Staubli VAL3: saveInputOutput.pjx

--- saveInputOutput.pjx ---
Parameters version=s7.5 stackSize=5000 millimeterUnit=true
Program file=decompose_num.pgx
Program file=decompose_wait.pgx
Program file=getItem_num.pgx
Program file=getSize_num.pgx
Program file=getValue_num.pgx
Program file=get_num.pgx
Program file=insert_aCOunt.pgx
Program file=insert_aIn.pgx
Program file=insert_aOutput.pgx
Program file=insert_cCount.pgx
Program file=insert_dIn.pgx
Program file=insert_dOut.pgx
Program file=replaceIO.pgx
Program file=resetAll.pgx
Program file=setInput.pgx
Program file=setOutput.pgx
Data file=saveInputOutput.dtx
Type name=aioItem path=Disk://kernel/template/aioItem/aioItem.pjx
Type name=dioItem path=Disk://kernel/template/dioItem/dioItem.pjx
Type name=countItem path=Disk://kernel/template/countItem/countItem.pjx

--- saveInputOutput.dtx ---
public aio MbAnaIn[4]
  [0] = {link=ModbusSrv-0\Modbus-Word\MbAnaIn[0]}
  [1] = {link=ModbusSrv-0\Modbus-Word\MbAnaIn[1]}
  [2] = {link=ModbusSrv-0\Modbus-Word\MbAnaIn[2]}
  [3] = {link=ModbusSrv-0\Modbus-Word\MbAnaIn[3]}
public aio MbAnaOut[4]
  [0] = {link=ModbusSrv-0\Modbus-Word\MbAnaOut[0]}
  [1] = {link=ModbusSrv-0\Modbus-Word\MbAnaOut[1]}
  [2] = {link=ModbusSrv-0\Modbus-Word\MbAnaOut[2]}
  [3] = {link=ModbusSrv-0\Modbus-Word\MbAnaOut[3]}
aio aNull
public aio aUser[10]
public aio aio_in
public aio aio_out
public aio cAin0 = {link=Can-Aio\%IB7}
public aio cAin1 = {link=Can-Aio\%IB23}
public aio cAin2 = {link=Can-Aio\%IB39}
public aio cAin3 = {link=Can-Aio\%IB55}
aio cAout0
aio cAout1
aio cAout2
aio cAout3
public aioItem aCount{}
public aioItem aInput{}
public aioItem aOutput{}
public bool bArmIO
public bool bBio
public bool bCS8
public bool bMio
public countItem cCount{}
  [num0]
    bool bActive = true
    bool bEnable = true
    num nCount
    string sID = "num0"
    string sName = "num0"
  [num1]
    bool bActive = true
    bool bEnable = true
    num nCount
    string sID = "num1"
    string sName = "num1"
  [num2]
    bool bActive = true
    bool bEnable = true
    num nCount
    string sID = "num2"
    string sName = "num2"
  [num3]
    bool bActive = true
    bool bEnable = true
    num nCount
    string sID = "num3"
    string sName = "num3"
  [num4]
    bool bActive = true
    bool bEnable = true
    num nCount
    string sID = "num4"
    string sName = "num4"
  [num5]
    bool bActive = true
    bool bEnable = true
    num nCount
    string sID = "num5"
    string sName = "num5"
  [num6]
    bool bActive = true
    bool bEnable = true
    num nCount
    string sID = "num6"
    string sName = "num6"
  [num7]
    bool bActive = true
    bool bEnable = true
    num nCount
    string sID = "num7"
    string sName = "num7"
  [num8]
    bool bActive = true
    bool bEnable = true
    num nCount
    string sID = "num8"
    string sName = "num8"
  [num9]
    bool bActive = true
    bool bEnable = true
    num nCount
    string sID = "num9"
    string sName = "num9"
public dio MbIn[100]
  [0] = {link=ModbusSrv-0\Modbus-Bit\MbIn[0]}
  [1] = {link=ModbusSrv-0\Modbus-Bit\MbIn[1]}
  [2] = {link=ModbusSrv-0\Modbus-Bit\MbIn[2]}
  [3] = {link=ModbusSrv-0\Modbus-Bit\MbIn[3]}
  [4] = {link=ModbusSrv-0\Modbus-Bit\MbIn[4]}
  [5] = {link=ModbusSrv-0\Modbus-Bit\MbIn[5]}
  [6] = {link=ModbusSrv-0\Modbus-Bit\MbIn[6]}
  [7] = {link=ModbusSrv-0\Modbus-Bit\MbIn[7]}
  [8] = {link=ModbusSrv-0\Modbus-Bit\MbIn[8]}
  [9] = {link=ModbusSrv-0\Modbus-Bit\MbIn[9]}
  [10] = {link=ModbusSrv-0\Modbus-Bit\MbIn[10]}
  [11] = {link=ModbusSrv-0\Modbus-Bit\MbIn[11]}
  [12] = {link=ModbusSrv-0\Modbus-Bit\MbIn[12]}
  [13] = {link=ModbusSrv-0\Modbus-Bit\MbIn[13]}
  [14] = {link=ModbusSrv-0\Modbus-Bit\MbIn[14]}
  [15] = {link=ModbusSrv-0\Modbus-Bit\MbIn[15]}
  [16] = {link=ModbusSrv-0\Modbus-Bit\MbIn[16]}
  [17] = {link=ModbusSrv-0\Modbus-Bit\MbIn[17]}
  [18] = {link=ModbusSrv-0\Modbus-Bit\MbIn[18]}
  [19] = {link=ModbusSrv-0\Modbus-Bit\MbIn[19]}
  [20] = {link=ModbusSrv-0\Modbus-Bit\MbIn[20]}
  [21] = {link=ModbusSrv-0\Modbus-Bit\MbIn[21]}
  [22] = {link=ModbusSrv-0\Modbus-Bit\MbIn[22]}
  [23] = {link=ModbusSrv-0\Modbus-Bit\MbIn[23]}
  [24] = {link=ModbusSrv-0\Modbus-Bit\MbIn[24]}
  [25] = {link=ModbusSrv-0\Modbus-Bit\MbIn[25]}
  [26] = {link=ModbusSrv-0\Modbus-Bit\MbIn[26]}
  [27] = {link=ModbusSrv-0\Modbus-Bit\MbIn[27]}
  [28] = {link=ModbusSrv-0\Modbus-Bit\MbIn[28]}
  [29] = {link=ModbusSrv-0\Modbus-Bit\MbIn[29]}
  [30] = {link=ModbusSrv-0\Modbus-Bit\MbIn[30]}
  [31] = {link=ModbusSrv-0\Modbus-Bit\MbIn[31]}
  [32] = {link=ModbusSrv-0\Modbus-Bit\MbIn[32]}
  [33] = {link=ModbusSrv-0\Modbus-Bit\MbIn[33]}
  [34] = {link=ModbusSrv-0\Modbus-Bit\MbIn[34]}
  [35] = {link=ModbusSrv-0\Modbus-Bit\MbIn[35]}
  [36] = {link=ModbusSrv-0\Modbus-Bit\MbIn[36]}
  [37] = {link=ModbusSrv-0\Modbus-Bit\MbIn[37]}
  [38] = {link=ModbusSrv-0\Modbus-Bit\MbIn[38]}
  [39] = {link=ModbusSrv-0\Modbus-Bit\MbIn[39]}
  [40] = {link=ModbusSrv-0\Modbus-Bit\MbIn[40]}
  [41] = {link=ModbusSrv-0\Modbus-Bit\MbIn[41]}
  [42] = {link=ModbusSrv-0\Modbus-Bit\MbIn[42]}
  [43] = {link=ModbusSrv-0\Modbus-Bit\MbIn[43]}
  [44] = {link=ModbusSrv-0\Modbus-Bit\MbIn[44]}
  [45] = {link=ModbusSrv-0\Modbus-Bit\MbIn[45]}
  [46] = {link=ModbusSrv-0\Modbus-Bit\MbIn[46]}
  [47] = {link=ModbusSrv-0\Modbus-Bit\MbIn[47]}
  [48] = {link=ModbusSrv-0\Modbus-Bit\MbIn[48]}
  [49] = {link=ModbusSrv-0\Modbus-Bit\MbIn[49]}
  [50] = {link=ModbusSrv-0\Modbus-Bit\MbIn[50]}
  [51] = {link=ModbusSrv-0\Modbus-Bit\MbIn[51]}
  [52] = {link=ModbusSrv-0\Modbus-Bit\MbIn[52]}
  [53] = {link=ModbusSrv-0\Modbus-Bit\MbIn[53]}
  [54] = {link=ModbusSrv-0\Modbus-Bit\MbIn[54]}
  [55] = {link=ModbusSrv-0\Modbus-Bit\MbIn[55]}
  [56] = {link=ModbusSrv-0\Modbus-Bit\MbIn[56]}
  [57] = {link=ModbusSrv-0\Modbus-Bit\MbIn[57]}
  [58] = {link=ModbusSrv-0\Modbus-Bit\MbIn[58]}
  [59] = {link=ModbusSrv-0\Modbus-Bit\MbIn[59]}
  [60] = {link=ModbusSrv-0\Modbus-Bit\MbIn[60]}
  [61] = {link=ModbusSrv-0\Modbus-Bit\MbIn[61]}
  [62] = {link=ModbusSrv-0\Modbus-Bit\MbIn[62]}
  [63] = {link=ModbusSrv-0\Modbus-Bit\MbIn[63]}
  [64] = {link=ModbusSrv-0\Modbus-Bit\MbIn[64]}
  [65] = {link=ModbusSrv-0\Modbus-Bit\MbIn[65]}
  [66] = {link=ModbusSrv-0\Modbus-Bit\MbIn[66]}
  [67] = {link=ModbusSrv-0\Modbus-Bit\MbIn[67]}
  [68] = {link=ModbusSrv-0\Modbus-Bit\MbIn[68]}
  [69] = {link=ModbusSrv-0\Modbus-Bit\MbIn[69]}
  [70] = {link=ModbusSrv-0\Modbus-Bit\MbIn[70]}
  [71] = {link=ModbusSrv-0\Modbus-Bit\MbIn[71]}
  [72] = {link=ModbusSrv-0\Modbus-Bit\MbIn[72]}
  [73] = {link=ModbusSrv-0\Modbus-Bit\MbIn[73]}
  [74] = {link=ModbusSrv-0\Modbus-Bit\MbIn[74]}
  [75] = {link=ModbusSrv-0\Modbus-Bit\MbIn[75]}
  [76] = {link=ModbusSrv-0\Modbus-Bit\MbIn[76]}
  [77] = {link=ModbusSrv-0\Modbus-Bit\MbIn[77]}
  [78] = {link=ModbusSrv-0\Modbus-Bit\MbIn[78]}
  [79] = {link=ModbusSrv-0\Modbus-Bit\MbIn[79]}
  [80] = {link=ModbusSrv-0\Modbus-Bit\MbIn[80]}
  [81] = {link=ModbusSrv-0\Modbus-Bit\MbIn[81]}
  [82] = {link=ModbusSrv-0\Modbus-Bit\MbIn[82]}
  [83] = {link=ModbusSrv-0\Modbus-Bit\MbIn[83]}
  [84] = {link=ModbusSrv-0\Modbus-Bit\MbIn[84]}
  [85] = {link=ModbusSrv-0\Modbus-Bit\MbIn[85]}
  [86] = {link=ModbusSrv-0\Modbus-Bit\MbIn[86]}
  [87] = {link=ModbusSrv-0\Modbus-Bit\MbIn[87]}
  [88] = {link=ModbusSrv-0\Modbus-Bit\MbIn[88]}
  [89] = {link=ModbusSrv-0\Modbus-Bit\MbIn[89]}
  [90] = {link=ModbusSrv-0\Modbus-Bit\MbIn[90]}
  [91] = {link=ModbusSrv-0\Modbus-Bit\MbIn[91]}
  [92] = {link=ModbusSrv-0\Modbus-Bit\MbIn[92]}
  [93] = {link=ModbusSrv-0\Modbus-Bit\MbIn[93]}
  [94] = {link=ModbusSrv-0\Modbus-Bit\MbIn[94]}
  [95] = {link=ModbusSrv-0\Modbus-Bit\MbIn[95]}
  [96] = {link=ModbusSrv-0\Modbus-Bit\MbIn[96]}
  [97] = {link=ModbusSrv-0\Modbus-Bit\MbIn[97]}
  [98] = {link=ModbusSrv-0\Modbus-Bit\MbIn[98]}
  [99] = {link=ModbusSrv-0\Modbus-Bit\MbIn[99]}
public dio MbOut[100]
  [0] = {link=ModbusSrv-0\Modbus-Bit\MbOut[0]}
  [1] = {link=ModbusSrv-0\Modbus-Bit\MbOut[1]}
  [2] = {link=ModbusSrv-0\Modbus-Bit\MbOut[2]}
  [3] = {link=ModbusSrv-0\Modbus-Bit\MbOut[3]}
  [4] = {link=ModbusSrv-0\Modbus-Bit\MbOut[4]}
  [5] = {link=ModbusSrv-0\Modbus-Bit\MbOut[5]}
  [6] = {link=ModbusSrv-0\Modbus-Bit\MbOut[6]}
  [7] = {link=ModbusSrv-0\Modbus-Bit\MbOut[7]}
  [8] = {link=ModbusSrv-0\Modbus-Bit\MbOut[8]}
  [9] = {link=ModbusSrv-0\Modbus-Bit\MbOut[9]}
  [10] = {link=ModbusSrv-0\Modbus-Bit\MbOut[10]}
  [11] = {link=ModbusSrv-0\Modbus-Bit\MbOut[11]}
  [12] = {link=ModbusSrv-0\Modbus-Bit\MbOut[12]}
  [13] = {link=ModbusSrv-0\Modbus-Bit\MbOut[13]}
  [14] = {link=ModbusSrv-0\Modbus-Bit\MbOut[14]}
  [15] = {link=ModbusSrv-0\Modbus-Bit\MbOut[15]}
  [16] = {link=ModbusSrv-0\Modbus-Bit\MbOut[16]}
  [17] = {link=ModbusSrv-0\Modbus-Bit\MbOut[17]}
  [18] = {link=ModbusSrv-0\Modbus-Bit\MbOut[18]}
  [19] = {link=ModbusSrv-0\Modbus-Bit\MbOut[19]}
  [20] = {link=ModbusSrv-0\Modbus-Bit\MbOut[20]}
  [21] = {link=ModbusSrv-0\Modbus-Bit\MbOut[21]}
  [22] = {link=ModbusSrv-0\Modbus-Bit\MbOut[22]}
  [23] = {link=ModbusSrv-0\Modbus-Bit\MbOut[23]}
  [24] = {link=ModbusSrv-0\Modbus-Bit\MbOut[24]}
  [25] = {link=ModbusSrv-0\Modbus-Bit\MbOut[25]}
  [26] = {link=ModbusSrv-0\Modbus-Bit\MbOut[26]}
  [27] = {link=ModbusSrv-0\Modbus-Bit\MbOut[27]}
  [28] = {link=ModbusSrv-0\Modbus-Bit\MbOut[28]}
  [29] = {link=ModbusSrv-0\Modbus-Bit\MbOut[29]}
  [30] = {link=ModbusSrv-0\Modbus-Bit\MbOut[30]}
  [31] = {link=ModbusSrv-0\Modbus-Bit\MbOut[31]}
  [32] = {link=ModbusSrv-0\Modbus-Bit\MbOut[32]}
  [33] = {link=ModbusSrv-0\Modbus-Bit\MbOut[33]}
  [34] = {link=ModbusSrv-0\Modbus-Bit\MbOut[34]}
  [35] = {link=ModbusSrv-0\Modbus-Bit\MbOut[35]}
  [36] = {link=ModbusSrv-0\Modbus-Bit\MbOut[36]}
  [37] = {link=ModbusSrv-0\Modbus-Bit\MbOut[37]}
  [38] = {link=ModbusSrv-0\Modbus-Bit\MbOut[38]}
  [39] = {link=ModbusSrv-0\Modbus-Bit\MbOut[39]}
  [40] = {link=ModbusSrv-0\Modbus-Bit\MbOut[40]}
  [41] = {link=ModbusSrv-0\Modbus-Bit\MbOut[41]}
  [42] = {link=ModbusSrv-0\Modbus-Bit\MbOut[42]}
  [43] = {link=ModbusSrv-0\Modbus-Bit\MbOut[43]}
  [44] = {link=ModbusSrv-0\Modbus-Bit\MbOut[44]}
  [45] = {link=ModbusSrv-0\Modbus-Bit\MbOut[45]}
  [46] = {link=ModbusSrv-0\Modbus-Bit\MbOut[46]}
  [47] = {link=ModbusSrv-0\Modbus-Bit\MbOut[47]}
  [48] = {link=ModbusSrv-0\Modbus-Bit\MbOut[48]}
  [49] = {link=ModbusSrv-0\Modbus-Bit\MbOut[49]}
  [50] = {link=ModbusSrv-0\Modbus-Bit\MbOut[50]}
  [51] = {link=ModbusSrv-0\Modbus-Bit\MbOut[51]}
  [52] = {link=ModbusSrv-0\Modbus-Bit\MbOut[52]}
  [53] = {link=ModbusSrv-0\Modbus-Bit\MbOut[53]}
  [54] = {link=ModbusSrv-0\Modbus-Bit\MbOut[54]}
  [55] = {link=ModbusSrv-0\Modbus-Bit\MbOut[55]}
  [56] = {link=ModbusSrv-0\Modbus-Bit\MbOut[56]}
  [57] = {link=ModbusSrv-0\Modbus-Bit\MbOut[57]}
  [58] = {link=ModbusSrv-0\Modbus-Bit\MbOut[58]}
  [59] = {link=ModbusSrv-0\Modbus-Bit\MbOut[59]}
  [60] = {link=ModbusSrv-0\Modbus-Bit\MbOut[60]}
  [61] = {link=ModbusSrv-0\Modbus-Bit\MbOut[61]}
  [62] = {link=ModbusSrv-0\Modbus-Bit\MbOut[62]}
  [63] = {link=ModbusSrv-0\Modbus-Bit\MbOut[63]}
  [64] = {link=ModbusSrv-0\Modbus-Bit\MbOut[64]}
  [65] = {link=ModbusSrv-0\Modbus-Bit\MbOut[65]}
  [66] = {link=ModbusSrv-0\Modbus-Bit\MbOut[66]}
  [67] = {link=ModbusSrv-0\Modbus-Bit\MbOut[67]}
  [68] = {link=ModbusSrv-0\Modbus-Bit\MbOut[68]}
  [69] = {link=ModbusSrv-0\Modbus-Bit\MbOut[69]}
  [70] = {link=ModbusSrv-0\Modbus-Bit\MbOut[70]}
  [71] = {link=ModbusSrv-0\Modbus-Bit\MbOut[71]}
  [72] = {link=ModbusSrv-0\Modbus-Bit\MbOut[72]}
  [73] = {link=ModbusSrv-0\Modbus-Bit\MbOut[73]}
  [74] = {link=ModbusSrv-0\Modbus-Bit\MbOut[74]}
  [75] = {link=ModbusSrv-0\Modbus-Bit\MbOut[75]}
  [76] = {link=ModbusSrv-0\Modbus-Bit\MbOut[76]}
  [77] = {link=ModbusSrv-0\Modbus-Bit\MbOut[77]}
  [78] = {link=ModbusSrv-0\Modbus-Bit\MbOut[78]}
  [79] = {link=ModbusSrv-0\Modbus-Bit\MbOut[79]}
  [80] = {link=ModbusSrv-0\Modbus-Bit\MbOut[80]}
  [81] = {link=ModbusSrv-0\Modbus-Bit\MbOut[81]}
  [82] = {link=ModbusSrv-0\Modbus-Bit\MbOut[82]}
  [83] = {link=ModbusSrv-0\Modbus-Bit\MbOut[83]}
  [84] = {link=ModbusSrv-0\Modbus-Bit\MbOut[84]}
  [85] = {link=ModbusSrv-0\Modbus-Bit\MbOut[85]}
  [86] = {link=ModbusSrv-0\Modbus-Bit\MbOut[86]}
  [87] = {link=ModbusSrv-0\Modbus-Bit\MbOut[87]}
  [88] = {link=ModbusSrv-0\Modbus-Bit\MbOut[88]}
  [89] = {link=ModbusSrv-0\Modbus-Bit\MbOut[89]}
  [90] = {link=ModbusSrv-0\Modbus-Bit\MbOut[90]}
  [91] = {link=ModbusSrv-0\Modbus-Bit\MbOut[91]}
  [92] = {link=ModbusSrv-0\Modbus-Bit\MbOut[92]}
  [93] = {link=ModbusSrv-0\Modbus-Bit\MbOut[93]}
  [94] = {link=ModbusSrv-0\Modbus-Bit\MbOut[94]}
  [95] = {link=ModbusSrv-0\Modbus-Bit\MbOut[95]}
  [96] = {link=ModbusSrv-0\Modbus-Bit\MbOut[96]}
  [97] = {link=ModbusSrv-0\Modbus-Bit\MbOut[97]}
  [98] = {link=ModbusSrv-0\Modbus-Bit\MbOut[98]}
  [99] = {link=ModbusSrv-0\Modbus-Bit\MbOut[99]}
dio NetIn0 = {link=ApplicomIO-1\TOPIC1_A-BLOCKA\%I0}
dio NetIn1 = {link=ApplicomIO-1\TOPIC1_A-BLOCKA\%I1}
dio NetIn10 = {link=ApplicomIO-1\TOPIC1_A-BLOCKA\%I10}
dio NetIn11 = {link=ApplicomIO-1\TOPIC1_A-BLOCKA\%I11}
dio NetIn12 = {link=ApplicomIO-1\TOPIC1_A-BLOCKA\%I12}
dio NetIn13 = {link=ApplicomIO-1\TOPIC1_A-BLOCKA\%I13}
dio NetIn14 = {link=ApplicomIO-1\TOPIC1_A-BLOCKA\%I14}
dio NetIn15 = {link=ApplicomIO-1\TOPIC1_A-BLOCKA\%I15}
dio NetIn16 = {link=ApplicomIO-1\TOPIC1_A-BLOCKA\%I16}
dio NetIn17 = {link=ApplicomIO-1\TOPIC1_A-BLOCKA\%I17}
dio NetIn18 = {link=ApplicomIO-1\TOPIC1_A-BLOCKA\%I18}
dio NetIn19 = {link=ApplicomIO-1\TOPIC1_A-BLOCKA\%I19}
dio NetIn2 = {link=ApplicomIO-1\TOPIC1_A-BLOCKA\%I2}
dio NetIn20 = {link=ApplicomIO-1\TOPIC1_A-BLOCKA\%I20}
dio NetIn21 = {link=ApplicomIO-1\TOPIC1_A-BLOCKA\%I21}
dio NetIn22 = {link=ApplicomIO-1\TOPIC1_A-BLOCKA\%I22}
dio NetIn23 = {link=ApplicomIO-1\TOPIC1_A-BLOCKA\%I23}
dio NetIn24 = {link=ApplicomIO-1\TOPIC1_A-BLOCKA\%I24}
dio NetIn25 = {link=ApplicomIO-1\TOPIC1_A-BLOCKA\%I25}
dio NetIn26 = {link=ApplicomIO-1\TOPIC1_A-BLOCKA\%I26}
dio NetIn27 = {link=ApplicomIO-1\TOPIC1_A-BLOCKA\%I27}
dio NetIn28 = {link=ApplicomIO-1\TOPIC1_A-BLOCKA\%I28}
dio NetIn29 = {link=ApplicomIO-1\TOPIC1_A-BLOCKA\%I29}
dio NetIn3 = {link=ApplicomIO-1\TOPIC1_A-BLOCKA\%I3}
dio NetIn30 = {link=ApplicomIO-1\TOPIC1_A-BLOCKA\%I30}
dio NetIn31 = {link=ApplicomIO-1\TOPIC1_A-BLOCKA\%I31}
dio NetIn32 = {link=ApplicomIO-1\TOPIC1_A-BLOCKA\%I32}
dio NetIn33 = {link=ApplicomIO-1\TOPIC1_A-BLOCKA\%I33}
dio NetIn34 = {link=ApplicomIO-1\TOPIC1_A-BLOCKA\%I34}
dio NetIn35 = {link=ApplicomIO-1\TOPIC1_A-BLOCKA\%I35}
dio NetIn36 = {link=ApplicomIO-1\TOPIC1_A-BLOCKA\%I36}
dio NetIn37 = {link=ApplicomIO-1\TOPIC1_A-BLOCKA\%I37}
dio NetIn38 = {link=ApplicomIO-1\TOPIC1_A-BLOCKA\%I38}
dio NetIn39 = {link=ApplicomIO-1\TOPIC1_A-BLOCKA\%I39}
dio NetIn4 = {link=ApplicomIO-1\TOPIC1_A-BLOCKA\%I4}
dio NetIn40 = {link=ApplicomIO-1\TOPIC1_A-BLOCKA\%I40}
dio NetIn41 = {link=ApplicomIO-1\TOPIC1_A-BLOCKA\%I41}
dio NetIn42 = {link=ApplicomIO-1\TOPIC1_A-BLOCKA\%I42}
dio NetIn43 = {link=ApplicomIO-1\TOPIC1_A-BLOCKA\%I43}
dio NetIn44 = {link=ApplicomIO-1\TOPIC1_A-BLOCKA\%I44}
dio NetIn45 = {link=ApplicomIO-1\TOPIC1_A-BLOCKA\%I45}
dio NetIn46 = {link=ApplicomIO-1\TOPIC1_A-BLOCKA\%I46}
dio NetIn47 = {link=ApplicomIO-1\TOPIC1_A-BLOCKA\%I47}
dio NetIn48 = {link=ApplicomIO-1\TOPIC1_A-BLOCKA\%I48}
dio NetIn49 = {link=ApplicomIO-1\TOPIC1_A-BLOCKA\%I49}
dio NetIn5 = {link=ApplicomIO-1\TOPIC1_A-BLOCKA\%I5}
dio NetIn50 = {link=ApplicomIO-1\TOPIC1_A-BLOCKA\%I50}
dio NetIn51 = {link=ApplicomIO-1\TOPIC1_A-BLOCKA\%I51}
dio NetIn52 = {link=ApplicomIO-1\TOPIC1_A-BLOCKA\%I52}
dio NetIn53 = {link=ApplicomIO-1\TOPIC1_A-BLOCKA\%I53}
dio NetIn54 = {link=ApplicomIO-1\TOPIC1_A-BLOCKA\%I54}
dio NetIn55 = {link=ApplicomIO-1\TOPIC1_A-BLOCKA\%I55}
dio NetIn56 = {link=ApplicomIO-1\TOPIC1_A-BLOCKA\%I56}
dio NetIn57 = {link=ApplicomIO-1\TOPIC1_A-BLOCKA\%I57}
dio NetIn58 = {link=ApplicomIO-1\TOPIC1_A-BLOCKA\%I58}
dio NetIn59 = {link=ApplicomIO-1\TOPIC1_A-BLOCKA\%I59}
dio NetIn6 = {link=ApplicomIO-1\TOPIC1_A-BLOCKA\%I6}
dio NetIn60 = {link=ApplicomIO-1\TOPIC1_A-BLOCKA\%I60}
dio NetIn61 = {link=ApplicomIO-1\TOPIC1_A-BLOCKA\%I61}
dio NetIn62 = {link=ApplicomIO-1\TOPIC1_A-BLOCKA\%I62}
dio NetIn63 = {link=ApplicomIO-1\TOPIC1_A-BLOCKA\%I63}
dio NetIn7 = {link=ApplicomIO-1\TOPIC1_A-BLOCKA\%I7}
dio NetIn8 = {link=ApplicomIO-1\TOPIC1_A-BLOCKA\%I8}
dio NetIn9 = {link=ApplicomIO-1\TOPIC1_A-BLOCKA\%I9}
dio NetOut0 = {link=ApplicomIO-1\TOPIC1_A-BLOCKA\%Q0}
dio NetOut1 = {link=ApplicomIO-1\TOPIC1_A-BLOCKA\%Q1}
dio NetOut10 = {link=ApplicomIO-1\TOPIC1_A-BLOCKA\%Q10}
dio NetOut11 = {link=ApplicomIO-1\TOPIC1_A-BLOCKA\%Q11}
dio NetOut12 = {link=ApplicomIO-1\TOPIC1_A-BLOCKA\%Q12}
dio NetOut13 = {link=ApplicomIO-1\TOPIC1_A-BLOCKA\%Q13}
dio NetOut14 = {link=ApplicomIO-1\TOPIC1_A-BLOCKA\%Q14}
dio NetOut15 = {link=ApplicomIO-1\TOPIC1_A-BLOCKA\%Q15}
dio NetOut16 = {link=ApplicomIO-1\TOPIC1_A-BLOCKA\%Q16}
dio NetOut17 = {link=ApplicomIO-1\TOPIC1_A-BLOCKA\%Q17}
dio NetOut18 = {link=ApplicomIO-1\TOPIC1_A-BLOCKA\%Q18}
dio NetOut19 = {link=ApplicomIO-1\TOPIC1_A-BLOCKA\%Q19}
dio NetOut2 = {link=ApplicomIO-1\TOPIC1_A-BLOCKA\%Q2}
dio NetOut20 = {link=ApplicomIO-1\TOPIC1_A-BLOCKA\%Q20}
dio NetOut21 = {link=ApplicomIO-1\TOPIC1_A-BLOCKA\%Q21}
dio NetOut22 = {link=ApplicomIO-1\TOPIC1_A-BLOCKA\%Q22}
dio NetOut23 = {link=ApplicomIO-1\TOPIC1_A-BLOCKA\%Q23}
dio NetOut24 = {link=ApplicomIO-1\TOPIC1_A-BLOCKA\%Q24}
dio NetOut25 = {link=ApplicomIO-1\TOPIC1_A-BLOCKA\%Q25}
dio NetOut26 = {link=ApplicomIO-1\TOPIC1_A-BLOCKA\%Q26}
dio NetOut27 = {link=ApplicomIO-1\TOPIC1_A-BLOCKA\%Q27}
dio NetOut28 = {link=ApplicomIO-1\TOPIC1_A-BLOCKA\%Q28}
dio NetOut29 = {link=ApplicomIO-1\TOPIC1_A-BLOCKA\%Q29}
dio NetOut3 = {link=ApplicomIO-1\TOPIC1_A-BLOCKA\%Q3}
dio NetOut30 = {link=ApplicomIO-1\TOPIC1_A-BLOCKA\%Q30}
dio NetOut31 = {link=ApplicomIO-1\TOPIC1_A-BLOCKA\%Q31}
dio NetOut32 = {link=ApplicomIO-1\TOPIC1_A-BLOCKA\%Q32}
dio NetOut33 = {link=ApplicomIO-1\TOPIC1_A-BLOCKA\%Q33}
dio NetOut34 = {link=ApplicomIO-1\TOPIC1_A-BLOCKA\%Q34}
dio NetOut35 = {link=ApplicomIO-1\TOPIC1_A-BLOCKA\%Q35}
dio NetOut36 = {link=ApplicomIO-1\TOPIC1_A-BLOCKA\%Q36}
dio NetOut37 = {link=ApplicomIO-1\TOPIC1_A-BLOCKA\%Q37}
dio NetOut38 = {link=ApplicomIO-1\TOPIC1_A-BLOCKA\%Q38}
dio NetOut39 = {link=ApplicomIO-1\TOPIC1_A-BLOCKA\%Q39}
dio NetOut4 = {link=ApplicomIO-1\TOPIC1_A-BLOCKA\%Q4}
dio NetOut40 = {link=ApplicomIO-1\TOPIC1_A-BLOCKA\%Q40}
dio NetOut41 = {link=ApplicomIO-1\TOPIC1_A-BLOCKA\%Q41}
dio NetOut42 = {link=ApplicomIO-1\TOPIC1_A-BLOCKA\%Q42}
dio NetOut43 = {link=ApplicomIO-1\TOPIC1_A-BLOCKA\%Q43}
dio NetOut44 = {link=ApplicomIO-1\TOPIC1_A-BLOCKA\%Q44}
dio NetOut45 = {link=ApplicomIO-1\TOPIC1_A-BLOCKA\%Q45}
dio NetOut46 = {link=ApplicomIO-1\TOPIC1_A-BLOCKA\%Q46}
dio NetOut47 = {link=ApplicomIO-1\TOPIC1_A-BLOCKA\%Q47}
dio NetOut48 = {link=ApplicomIO-1\TOPIC1_A-BLOCKA\%Q48}
dio NetOut49 = {link=ApplicomIO-1\TOPIC1_A-BLOCKA\%Q49}
dio NetOut5 = {link=ApplicomIO-1\TOPIC1_A-BLOCKA\%Q5}
dio NetOut50 = {link=ApplicomIO-1\TOPIC1_A-BLOCKA\%Q50}
dio NetOut51 = {link=ApplicomIO-1\TOPIC1_A-BLOCKA\%Q51}
dio NetOut52 = {link=ApplicomIO-1\TOPIC1_A-BLOCKA\%Q52}
dio NetOut53 = {link=ApplicomIO-1\TOPIC1_A-BLOCKA\%Q53}
dio NetOut54 = {link=ApplicomIO-1\TOPIC1_A-BLOCKA\%Q54}
dio NetOut55 = {link=ApplicomIO-1\TOPIC1_A-BLOCKA\%Q55}
dio NetOut56 = {link=ApplicomIO-1\TOPIC1_A-BLOCKA\%Q56}
dio NetOut57 = {link=ApplicomIO-1\TOPIC1_A-BLOCKA\%Q57}
dio NetOut58 = {link=ApplicomIO-1\TOPIC1_A-BLOCKA\%Q58}
dio NetOut59 = {link=ApplicomIO-1\TOPIC1_A-BLOCKA\%Q59}
dio NetOut6 = {link=ApplicomIO-1\TOPIC1_A-BLOCKA\%Q6}
dio NetOut60 = {link=ApplicomIO-1\TOPIC1_A-BLOCKA\%Q60}
dio NetOut61 = {link=ApplicomIO-1\TOPIC1_A-BLOCKA\%Q61}
dio NetOut62 = {link=ApplicomIO-1\TOPIC1_A-BLOCKA\%Q62}
dio NetOut63 = {link=ApplicomIO-1\TOPIC1_A-BLOCKA\%Q63}
dio NetOut7 = {link=ApplicomIO-1\TOPIC1_A-BLOCKA\%Q7}
dio NetOut8 = {link=ApplicomIO-1\TOPIC1_A-BLOCKA\%Q8}
dio NetOut9 = {link=ApplicomIO-1\TOPIC1_A-BLOCKA\%Q9}
public dio b2In0 = {link=BasicIO-2\%I0}
public dio b2In1 = {link=BasicIO-2\%I1}
public dio b2In10 = {link=BasicIO-2\%I10}
public dio b2In11 = {link=BasicIO-2\%I11}
public dio b2In12 = {link=BasicIO-2\%I12}
public dio b2In13 = {link=BasicIO-2\%I13}
public dio b2In14 = {link=BasicIO-2\%I14}
public dio b2In15 = {link=BasicIO-2\%I15}
public dio b2In2 = {link=BasicIO-2\%I2}
public dio b2In3 = {link=BasicIO-2\%I3}
public dio b2In4 = {link=BasicIO-2\%I4}
public dio b2In5 = {link=BasicIO-2\%I5}
public dio b2In6 = {link=BasicIO-2\%I6}
public dio b2In7 = {link=BasicIO-2\%I7}
public dio b2In8 = {link=BasicIO-2\%I8}
public dio b2In9 = {link=BasicIO-2\%I9}
public dio b2Out0 = {link=BasicIO-2\%Q0}
public dio b2Out1 = {link=BasicIO-2\%Q1}
public dio b2Out10 = {link=BasicIO-2\%Q10}
public dio b2Out11 = {link=BasicIO-2\%Q11}
public dio b2Out12 = {link=BasicIO-2\%Q12}
public dio b2Out13 = {link=BasicIO-2\%Q13}
public dio b2Out14 = {link=BasicIO-2\%Q14}
public dio b2Out15 = {link=BasicIO-2\%Q15}
public dio b2Out2 = {link=BasicIO-2\%Q2}
public dio b2Out3 = {link=BasicIO-2\%Q3}
public dio b2Out4 = {link=BasicIO-2\%Q4}
public dio b2Out5 = {link=BasicIO-2\%Q5}
public dio b2Out6 = {link=BasicIO-2\%Q6}
public dio b2Out7 = {link=BasicIO-2\%Q7}
public dio b2Out8 = {link=BasicIO-2\%Q8}
public dio b2Out9 = {link=BasicIO-2\%Q9}
public dio bIn0 = {link=BasicIO-1\%I0}
public dio bIn1 = {link=BasicIO-1\%I1}
public dio bIn10 = {link=BasicIO-1\%I10}
public dio bIn11 = {link=BasicIO-1\%I11}
public dio bIn12 = {link=BasicIO-1\%I12}
public dio bIn13 = {link=BasicIO-1\%I13}
public dio bIn14 = {link=BasicIO-1\%I14}
public dio bIn15 = {link=BasicIO-1\%I15}
public dio bIn2 = {link=BasicIO-1\%I2}
public dio bIn3 = {link=BasicIO-1\%I3}
public dio bIn4 = {link=BasicIO-1\%I4}
public dio bIn5 = {link=BasicIO-1\%I5}
public dio bIn6 = {link=BasicIO-1\%I6}
public dio bIn7 = {link=BasicIO-1\%I7}
public dio bIn8 = {link=BasicIO-1\%I8}
public dio bIn9 = {link=BasicIO-1\%I9}
public dio bOut0 = {link=BasicIO-1\%Q0}
public dio bOut1 = {link=BasicIO-1\%Q1}
public dio bOut10 = {link=BasicIO-1\%Q10}
public dio bOut11 = {link=BasicIO-1\%Q11}
public dio bOut12 = {link=BasicIO-1\%Q12}
public dio bOut13 = {link=BasicIO-1\%Q13}
public dio bOut14 = {link=BasicIO-1\%Q14}
public dio bOut15 = {link=BasicIO-1\%Q15}
public dio bOut2 = {link=BasicIO-1\%Q2}
public dio bOut3 = {link=BasicIO-1\%Q3}
public dio bOut4 = {link=BasicIO-1\%Q4}
public dio bOut5 = {link=BasicIO-1\%Q5}
public dio bOut6 = {link=BasicIO-1\%Q6}
public dio bOut7 = {link=BasicIO-1\%Q7}
public dio bOut8 = {link=BasicIO-1\%Q8}
public dio bOut9 = {link=BasicIO-1\%Q9}
public dio cDin0 = {link=Can-Dio\%I0}
public dio cDin1 = {link=Can-Dio\%I1}
public dio cDin2 = {link=Can-Dio\%I2}
public dio cDin3 = {link=Can-Dio\%I3}
public dio cDin4 = {link=Can-Dio\%I4}
public dio cDin5 = {link=Can-Dio\%I5}
public dio cDin6 = {link=Can-Dio\%I6}
public dio cDin7 = {link=Can-Dio\%I7}
public dio cDout0 = {link=Can-Dio\%Q0}
public dio cDout1 = {link=Can-Dio\%Q1}
public dio cDout2 = {link=Can-Dio\%Q2}
public dio cDout3 = {link=Can-Dio\%Q3}
public dio cDout4 = {link=Can-Dio\%Q4}
public dio cDout5 = {link=Can-Dio\%Q5}
public dio cDout6 = {link=Can-Dio\%Q6}
public dio cDout7 = {link=Can-Dio\%Q7}
public dio dInUser
dio dNull
public dio dOutUser
public dio fIn0 = {link=fIn0}
public dio fIn1 = {link=fIn1}
public dio fOut0 = {link=fOut0}
public dio mIn0 = {link=ModuleIO\%I0}
public dio mIn1 = {link=ModuleIO\%I1}
public dio mIn10 = {link=ModuleIO\%I10}
public dio mIn11 = {link=ModuleIO\%I11}
public dio mIn12 = {link=ModuleIO\%I12}
public dio mIn13 = {link=ModuleIO\%I13}
public dio mIn14 = {link=ModuleIO\%I14}
public dio mIn15 = {link=ModuleIO\%I15}
public dio mIn16 = {link=ModuleIO\%I16}
public dio mIn17 = {link=ModuleIO\%I17}
public dio mIn18 = {link=ModuleIO\%I18}
public dio mIn19 = {link=ModuleIO\%I19}
public dio mIn2 = {link=ModuleIO\%I2}
public dio mIn20 = {link=ModuleIO\%I20}
public dio mIn21 = {link=ModuleIO\%I21}
public dio mIn22 = {link=ModuleIO\%I22}
public dio mIn23 = {link=ModuleIO\%I23}
public dio mIn24 = {link=ModuleIO\%I24}
public dio mIn25 = {link=ModuleIO\%I25}
public dio mIn26 = {link=ModuleIO\%I26}
public dio mIn27 = {link=ModuleIO\%I27}
public dio mIn28 = {link=ModuleIO\%I28}
public dio mIn29 = {link=ModuleIO\%I29}
public dio mIn3 = {link=ModuleIO\%I3}
public dio mIn30 = {link=ModuleIO\%I30}
public dio mIn31 = {link=ModuleIO\%I31}
public dio mIn4 = {link=ModuleIO\%I4}
public dio mIn5 = {link=ModuleIO\%I5}
public dio mIn6 = {link=ModuleIO\%I6}
public dio mIn7 = {link=ModuleIO\%I7}
public dio mIn8 = {link=ModuleIO\%I8}
public dio mIn9 = {link=ModuleIO\%I9}
public dio mOut0 = {link=ModuleIO\%Q0}
public dio mOut1 = {link=ModuleIO\%Q1}
public dio mOut10 = {link=ModuleIO\%Q10}
public dio mOut11 = {link=ModuleIO\%Q11}
public dio mOut12 = {link=ModuleIO\%Q12}
public dio mOut13 = {link=ModuleIO\%Q13}
public dio mOut14 = {link=ModuleIO\%Q14}
public dio mOut15 = {link=ModuleIO\%Q15}
public dio mOut16 = {link=ModuleIO\%Q16}
public dio mOut17 = {link=ModuleIO\%Q17}
public dio mOut18 = {link=ModuleIO\%Q18}
public dio mOut19 = {link=ModuleIO\%Q19}
public dio mOut2 = {link=ModuleIO\%Q2}
public dio mOut20 = {link=ModuleIO\%Q20}
public dio mOut21 = {link=ModuleIO\%Q21}
public dio mOut22 = {link=ModuleIO\%Q22}
public dio mOut23 = {link=ModuleIO\%Q23}
public dio mOut24 = {link=ModuleIO\%Q24}
public dio mOut25 = {link=ModuleIO\%Q25}
public dio mOut26 = {link=ModuleIO\%Q26}
public dio mOut27 = {link=ModuleIO\%Q27}
public dio mOut28 = {link=ModuleIO\%Q28}
public dio mOut29 = {link=ModuleIO\%Q29}
public dio mOut3 = {link=ModuleIO\%Q3}
public dio mOut30 = {link=ModuleIO\%Q30}
public dio mOut31 = {link=ModuleIO\%Q31}
public dio mOut4 = {link=ModuleIO\%Q4}
public dio mOut5 = {link=ModuleIO\%Q5}
public dio mOut6 = {link=ModuleIO\%Q6}
public dio mOut7 = {link=ModuleIO\%Q7}
public dio mOut8 = {link=ModuleIO\%Q8}
public dio mOut9 = {link=ModuleIO\%Q9}
public dio usrIn0 = {link=usrIn0}
public dio usrIn1 = {link=usrIn1}
public dio valve1 = {link=valve1}
public dio valve2 = {link=valve2}
public dioItem dInput{}
  [NetIn00]
    bool bActive
    bool bEnable = true
    dio dDio = {link=ApplicomIO-1\TOPIC1_A-BLOCKA\%I0}
    string sID = "NetIn00"
    string sName = "NetIn00"
  [NetIn01]
    bool bActive
    bool bEnable = true
    dio dDio = {link=ApplicomIO-1\TOPIC1_A-BLOCKA\%I1}
    string sID = "NetIn01"
    string sName = "NetIn01"
  [NetIn02]
    bool bActive
    bool bEnable = true
    dio dDio = {link=ApplicomIO-1\TOPIC1_A-BLOCKA\%I2}
    string sID = "NetIn02"
    string sName = "NetIn02"
  [NetIn03]
    bool bActive
    bool bEnable = true
    dio dDio = {link=ApplicomIO-1\TOPIC1_A-BLOCKA\%I3}
    string sID = "NetIn03"
    string sName = "NetIn03"
  [NetIn04]
    bool bActive
    bool bEnable = true
    dio dDio = {link=ApplicomIO-1\TOPIC1_A-BLOCKA\%I4}
    string sID = "NetIn04"
    string sName = "NetIn04"
  [NetIn05]
    bool bActive
    bool bEnable = true
    dio dDio = {link=ApplicomIO-1\TOPIC1_A-BLOCKA\%I5}
    string sID = "NetIn05"
    string sName = "NetIn05"
  [NetIn06]
    bool bActive
    bool bEnable = true
    dio dDio = {link=ApplicomIO-1\TOPIC1_A-BLOCKA\%I6}
    string sID = "NetIn06"
    string sName = "NetIn06"
  [NetIn07]
    bool bActive
    bool bEnable = true
    dio dDio = {link=ApplicomIO-1\TOPIC1_A-BLOCKA\%I7}
    string sID = "NetIn07"
    string sName = "NetIn07"
  [NetIn08]
    bool bActive
    bool bEnable = true
    dio dDio = {link=ApplicomIO-1\TOPIC1_A-BLOCKA\%I8}
    string sID = "NetIn08"
    string sName = "NetIn08"
  [NetIn09]
    bool bActive
    bool bEnable = true
    dio dDio = {link=ApplicomIO-1\TOPIC1_A-BLOCKA\%I9}
    string sID = "NetIn09"
    string sName = "NetIn09"
  [NetIn10]
    bool bActive
    bool bEnable = true
    dio dDio = {link=ApplicomIO-1\TOPIC1_A-BLOCKA\%I10}
    string sID = "NetIn10"
    string sName = "NetIn10"
  [NetIn11]
    bool bActive
    bool bEnable = true
    dio dDio = {link=ApplicomIO-1\TOPIC1_A-BLOCKA\%I11}
    string sID = "NetIn11"
    string sName = "NetIn11"
  [NetIn12]
    bool bActive
    bool bEnable = true
    dio dDio = {link=ApplicomIO-1\TOPIC1_A-BLOCKA\%I12}
    string sID = "NetIn12"
    string sName = "NetIn12"
  [NetIn13]
    bool bActive
    bool bEnable = true
    dio dDio = {link=ApplicomIO-1\TOPIC1_A-BLOCKA\%I13}
    string sID = "NetIn13"
    string sName = "NetIn13"
  [NetIn14]
    bool bActive
    bool bEnable = true
    dio dDio = {link=ApplicomIO-1\TOPIC1_A-BLOCKA\%I14}
    string sID = "NetIn14"
    string sName = "NetIn14"
  [NetIn15]
    bool bActive
    bool bEnable = true
    dio dDio = {link=ApplicomIO-1\TOPIC1_A-BLOCKA\%I15}
    string sID = "NetIn15"
    string sName = "NetIn15"
  [NetIn16]
    bool bActive
    bool bEnable = true
    dio dDio = {link=ApplicomIO-1\TOPIC1_A-BLOCKA\%I16}
    string sID = "NetIn16"
    string sName = "NetIn16"
  [NetIn17]
    bool bActive
    bool bEnable = true
    dio dDio = {link=ApplicomIO-1\TOPIC1_A-BLOCKA\%I17}
    string sID = "NetIn17"
    string sName = "NetIn17"
  [NetIn18]
    bool bActive
    bool bEnable = true
    dio dDio = {link=ApplicomIO-1\TOPIC1_A-BLOCKA\%I18}
    string sID = "NetIn18"
    string sName = "NetIn18"
  [NetIn19]
    bool bActive
    bool bEnable = true
    dio dDio = {link=ApplicomIO-1\TOPIC1_A-BLOCKA\%I19}
    string sID = "NetIn19"
    string sName = "NetIn19"
  [NetIn20]
    bool bActive
    bool bEnable = true
    dio dDio = {link=ApplicomIO-1\TOPIC1_A-BLOCKA\%I20}
    string sID = "NetIn20"
    string sName = "NetIn20"
  [NetIn21]
    bool bActive
    bool bEnable = true
    dio dDio = {link=ApplicomIO-1\TOPIC1_A-BLOCKA\%I21}
    string sID = "NetIn21"
    string sName = "NetIn21"
  [NetIn22]
    bool bActive
    bool bEnable = true
    dio dDio = {link=ApplicomIO-1\TOPIC1_A-BLOCKA\%I22}
    string sID = "NetIn22"
    string sName = "NetIn22"
  [NetIn23]
    bool bActive
    bool bEnable = true
    dio dDio = {link=ApplicomIO-1\TOPIC1_A-BLOCKA\%I23}
    string sID = "NetIn23"
    string sName = "NetIn23"
  [NetIn24]
    bool bActive
    bool bEnable = true
    dio dDio = {link=ApplicomIO-1\TOPIC1_A-BLOCKA\%I24}
    string sID = "NetIn24"
    string sName = "NetIn24"
  [NetIn25]
    bool bActive
    bool bEnable = true
    dio dDio = {link=ApplicomIO-1\TOPIC1_A-BLOCKA\%I25}
    string sID = "NetIn25"
    string sName = "NetIn25"
  [NetIn26]
    bool bActive
    bool bEnable = true
    dio dDio = {link=ApplicomIO-1\TOPIC1_A-BLOCKA\%I26}
    string sID = "NetIn26"
    string sName = "NetIn26"
  [NetIn27]
    bool bActive
    bool bEnable = true
    dio dDio = {link=ApplicomIO-1\TOPIC1_A-BLOCKA\%I27}
    string sID = "NetIn27"
    string sName = "NetIn27"
  [NetIn28]
    bool bActive
    bool bEnable = true
    dio dDio = {link=ApplicomIO-1\TOPIC1_A-BLOCKA\%I28}
    string sID = "NetIn28"
    string sName = "NetIn28"
  [NetIn29]
    bool bActive
    bool bEnable = true
    dio dDio = {link=ApplicomIO-1\TOPIC1_A-BLOCKA\%I29}
    string sID = "NetIn29"
    string sName = "NetIn29"
  [NetIn30]
    bool bActive
    bool bEnable = true
    dio dDio = {link=ApplicomIO-1\TOPIC1_A-BLOCKA\%I30}
    string sID = "NetIn30"
    string sName = "NetIn30"
  [NetIn31]
    bool bActive
    bool bEnable = true
    dio dDio = {link=ApplicomIO-1\TOPIC1_A-BLOCKA\%I31}
    string sID = "NetIn31"
    string sName = "NetIn31"
  [NetIn32]
    bool bActive
    bool bEnable = true
    dio dDio = {link=ApplicomIO-1\TOPIC1_A-BLOCKA\%I32}
    string sID = "NetIn32"
    string sName = "NetIn32"
  [NetIn33]
    bool bActive
    bool bEnable = true
    dio dDio = {link=ApplicomIO-1\TOPIC1_A-BLOCKA\%I33}
    string sID = "NetIn33"
    string sName = "NetIn33"
  [NetIn34]
    bool bActive
    bool bEnable = true
    dio dDio = {link=ApplicomIO-1\TOPIC1_A-BLOCKA\%I34}
    string sID = "NetIn34"
    string sName = "NetIn34"
  [NetIn35]
    bool bActive
    bool bEnable = true
    dio dDio = {link=ApplicomIO-1\TOPIC1_A-BLOCKA\%I35}
    string sID = "NetIn35"
    string sName = "NetIn35"
  [NetIn36]
    bool bActive
    bool bEnable = true
    dio dDio = {link=ApplicomIO-1\TOPIC1_A-BLOCKA\%I36}
    string sID = "NetIn36"
    string sName = "NetIn36"
  [NetIn37]
    bool bActive
    bool bEnable = true
    dio dDio = {link=ApplicomIO-1\TOPIC1_A-BLOCKA\%I37}
    string sID = "NetIn37"
    string sName = "NetIn37"
  [NetIn38]
    bool bActive
    bool bEnable = true
    dio dDio = {link=ApplicomIO-1\TOPIC1_A-BLOCKA\%I38}
    string sID = "NetIn38"
    string sName = "NetIn38"
  [NetIn39]
    bool bActive
    bool bEnable = true
    dio dDio = {link=ApplicomIO-1\TOPIC1_A-BLOCKA\%I39}
    string sID = "NetIn39"
    string sName = "NetIn39"
  [NetIn40]
    bool bActive
    bool bEnable = true
    dio dDio = {link=ApplicomIO-1\TOPIC1_A-BLOCKA\%I40}
    string sID = "NetIn40"
    string sName = "NetIn40"
  [NetIn41]
    bool bActive
    bool bEnable = true
    dio dDio = {link=ApplicomIO-1\TOPIC1_A-BLOCKA\%I41}
    string sID = "NetIn41"
    string sName = "NetIn41"
  [NetIn42]
    bool bActive
    bool bEnable = true
    dio dDio = {link=ApplicomIO-1\TOPIC1_A-BLOCKA\%I42}
    string sID = "NetIn42"
    string sName = "NetIn42"
  [NetIn43]
    bool bActive
    bool bEnable = true
    dio dDio = {link=ApplicomIO-1\TOPIC1_A-BLOCKA\%I43}
    string sID = "NetIn43"
    string sName = "NetIn43"
  [NetIn44]
    bool bActive
    bool bEnable = true
    dio dDio = {link=ApplicomIO-1\TOPIC1_A-BLOCKA\%I44}
    string sID = "NetIn44"
    string sName = "NetIn44"
  [NetIn45]
    bool bActive
    bool bEnable = true
    dio dDio = {link=ApplicomIO-1\TOPIC1_A-BLOCKA\%I45}
    string sID = "NetIn45"
    string sName = "NetIn45"
  [NetIn46]
    bool bActive
    bool bEnable = true
    dio dDio = {link=ApplicomIO-1\TOPIC1_A-BLOCKA\%I46}
    string sID = "NetIn46"
    string sName = "NetIn46"
  [NetIn47]
    bool bActive
    bool bEnable = true
    dio dDio = {link=ApplicomIO-1\TOPIC1_A-BLOCKA\%I47}
    string sID = "NetIn47"
    string sName = "NetIn47"
  [NetIn48]
    bool bActive
    bool bEnable = true
    dio dDio = {link=ApplicomIO-1\TOPIC1_A-BLOCKA\%I48}
    string sID = "NetIn48"
    string sName = "NetIn48"
  [NetIn49]
    bool bActive
    bool bEnable = true
    dio dDio = {link=ApplicomIO-1\TOPIC1_A-BLOCKA\%I49}
    string sID = "NetIn49"
    string sName = "NetIn49"
  [NetIn50]
    bool bActive
    bool bEnable = true
    dio dDio = {link=ApplicomIO-1\TOPIC1_A-BLOCKA\%I50}
    string sID = "NetIn50"
    string sName = "NetIn50"
  [NetIn51]
    bool bActive
    bool bEnable = true
    dio dDio = {link=ApplicomIO-1\TOPIC1_A-BLOCKA\%I51}
    string sID = "NetIn51"
    string sName = "NetIn51"
  [NetIn52]
    bool bActive
    bool bEnable = true
    dio dDio = {link=ApplicomIO-1\TOPIC1_A-BLOCKA\%I52}
    string sID = "NetIn52"
    string sName = "NetIn52"
  [NetIn53]
    bool bActive
    bool bEnable = true
    dio dDio = {link=ApplicomIO-1\TOPIC1_A-BLOCKA\%I53}
    string sID = "NetIn53"
    string sName = "NetIn53"
  [NetIn54]
    bool bActive
    bool bEnable = true
    dio dDio = {link=ApplicomIO-1\TOPIC1_A-BLOCKA\%I54}
    string sID = "NetIn54"
    string sName = "NetIn54"
  [NetIn55]
    bool bActive
    bool bEnable = true
    dio dDio = {link=ApplicomIO-1\TOPIC1_A-BLOCKA\%I55}
    string sID = "NetIn55"
    string sName = "NetIn55"
  [NetIn56]
    bool bActive
    bool bEnable = true
    dio dDio = {link=ApplicomIO-1\TOPIC1_A-BLOCKA\%I56}
    string sID = "NetIn56"
    string sName = "NetIn56"
  [NetIn57]
    bool bActive
    bool bEnable = true
    dio dDio = {link=ApplicomIO-1\TOPIC1_A-BLOCKA\%I57}
    string sID = "NetIn57"
    string sName = "NetIn57"
  [NetIn58]
    bool bActive
    bool bEnable = true
    dio dDio = {link=ApplicomIO-1\TOPIC1_A-BLOCKA\%I58}
    string sID = "NetIn58"
    string sName = "NetIn58"
  [NetIn59]
    bool bActive
    bool bEnable = true
    dio dDio = {link=ApplicomIO-1\TOPIC1_A-BLOCKA\%I59}
    string sID = "NetIn59"
    string sName = "NetIn59"
  [NetIn60]
    bool bActive
    bool bEnable = true
    dio dDio = {link=ApplicomIO-1\TOPIC1_A-BLOCKA\%I60}
    string sID = "NetIn60"
    string sName = "NetIn60"
  [NetIn61]
    bool bActive
    bool bEnable = true
    dio dDio = {link=ApplicomIO-1\TOPIC1_A-BLOCKA\%I61}
    string sID = "NetIn61"
    string sName = "NetIn61"
  [NetIn62]
    bool bActive
    bool bEnable = true
    dio dDio = {link=ApplicomIO-1\TOPIC1_A-BLOCKA\%I62}
    string sID = "NetIn62"
    string sName = "NetIn62"
  [NetIn63]
    bool bActive
    bool bEnable = true
    dio dDio = {link=ApplicomIO-1\TOPIC1_A-BLOCKA\%I63}
    string sID = "NetIn63"
    string sName = "NetIn63"
  [fIn0]
    bool bActive = true
    bool bEnable = true
    dio dDio = {link=fIn0}
    string sID = "fIn0"
    string sName = "fIn0"
  [fIn1]
    bool bActive = true
    bool bEnable = true
    dio dDio = {link=fIn1}
    string sID = "fIn1"
    string sName = "fIn1"
  [usrIn0]
    bool bActive = true
    bool bEnable = true
    dio dDio = {link=usrIn0}
    string sID = "usrIn0"
    string sName = "usrIn0"
  [usrIn1]
    bool bActive = true
    bool bEnable = true
    dio dDio = {link=usrIn1}
    string sID = "usrIn1"
    string sName = "usrIn1"
public dioItem dOutput{}
  [NetOut00]
    bool bActive
    bool bEnable = true
    dio dDio = {link=ApplicomIO-1\TOPIC1_A-BLOCKA\%Q0}
    string sID = "NetOut00"
    string sName = "NetOut00"
  [NetOut01]
    bool bActive
    bool bEnable = true
    dio dDio = {link=ApplicomIO-1\TOPIC1_A-BLOCKA\%Q1}
    string sID = "NetOut01"
    string sName = "NetOut01"
  [NetOut02]
    bool bActive
    bool bEnable = true
    dio dDio = {link=ApplicomIO-1\TOPIC1_A-BLOCKA\%Q2}
    string sID = "NetOut02"
    string sName = "NetOut02"
  [NetOut03]
    bool bActive
    bool bEnable = true
    dio dDio = {link=ApplicomIO-1\TOPIC1_A-BLOCKA\%Q3}
    string sID = "NetOut03"
    string sName = "NetOut03"
  [NetOut04]
    bool bActive
    bool bEnable = true
    dio dDio = {link=ApplicomIO-1\TOPIC1_A-BLOCKA\%Q4}
    string sID = "NetOut04"
    string sName = "NetOut04"
  [NetOut05]
    bool bActive
    bool bEnable = true
    dio dDio = {link=ApplicomIO-1\TOPIC1_A-BLOCKA\%Q5}
    string sID = "NetOut05"
    string sName = "NetOut05"
  [NetOut06]
    bool bActive
    bool bEnable = true
    dio dDio = {link=ApplicomIO-1\TOPIC1_A-BLOCKA\%Q6}
    string sID = "NetOut06"
    string sName = "NetOut06"
  [NetOut07]
    bool bActive
    bool bEnable = true
    dio dDio = {link=ApplicomIO-1\TOPIC1_A-BLOCKA\%Q7}
    string sID = "NetOut07"
    string sName = "NetOut07"
  [NetOut08]
    bool bActive
    bool bEnable = true
    dio dDio = {link=ApplicomIO-1\TOPIC1_A-BLOCKA\%Q8}
    string sID = "NetOut08"
    string sName = "NetOut08"
  [NetOut09]
    bool bActive
    bool bEnable = true
    dio dDio = {link=ApplicomIO-1\TOPIC1_A-BLOCKA\%Q9}
    string sID = "NetOut09"
    string sName = "NetOut09"
  [NetOut10]
    bool bActive
    bool bEnable = true
    dio dDio = {link=ApplicomIO-1\TOPIC1_A-BLOCKA\%Q10}
    string sID = "NetOut10"
    string sName = "NetOut10"
  [NetOut11]
    bool bActive
    bool bEnable = true
    dio dDio = {link=ApplicomIO-1\TOPIC1_A-BLOCKA\%Q11}
    string sID = "NetOut11"
    string sName = "NetOut11"
  [NetOut12]
    bool bActive
    bool bEnable = true
    dio dDio = {link=ApplicomIO-1\TOPIC1_A-BLOCKA\%Q12}
    string sID = "NetOut12"
    string sName = "NetOut12"
  [NetOut13]
    bool bActive
    bool bEnable = true
    dio dDio = {link=ApplicomIO-1\TOPIC1_A-BLOCKA\%Q13}
    string sID = "NetOut13"
    string sName = "NetOut13"
  [NetOut14]
    bool bActive
    bool bEnable = true
    dio dDio = {link=ApplicomIO-1\TOPIC1_A-BLOCKA\%Q14}
    string sID = "NetOut14"
    string sName = "NetOut14"
  [NetOut15]
    bool bActive
    bool bEnable = true
    dio dDio = {link=ApplicomIO-1\TOPIC1_A-BLOCKA\%Q15}
    string sID = "NetOut15"
    string sName = "NetOut15"
  [NetOut16]
    bool bActive
    bool bEnable = true
    dio dDio = {link=ApplicomIO-1\TOPIC1_A-BLOCKA\%Q16}
    string sID = "NetOut16"
    string sName = "NetOut16"
  [NetOut17]
    bool bActive
    bool bEnable = true
    dio dDio = {link=ApplicomIO-1\TOPIC1_A-BLOCKA\%Q17}
    string sID = "NetOut17"
    string sName = "NetOut17"
  [NetOut18]
    bool bActive
    bool bEnable = true
    dio dDio = {link=ApplicomIO-1\TOPIC1_A-BLOCKA\%Q18}
    string sID = "NetOut18"
    string sName = "NetOut18"
  [NetOut19]
    bool bActive
    bool bEnable = true
    dio dDio = {link=ApplicomIO-1\TOPIC1_A-BLOCKA\%Q19}
    string sID = "NetOut19"
    string sName = "NetOut19"
  [NetOut20]
    bool bActive
    bool bEnable = true
    dio dDio = {link=ApplicomIO-1\TOPIC1_A-BLOCKA\%Q20}
    string sID = "NetOut20"
    string sName = "NetOut20"
  [NetOut21]
    bool bActive
    bool bEnable = true
    dio dDio = {link=ApplicomIO-1\TOPIC1_A-BLOCKA\%Q21}
    string sID = "NetOut21"
    string sName = "NetOut21"
  [NetOut22]
    bool bActive
    bool bEnable = true
    dio dDio = {link=ApplicomIO-1\TOPIC1_A-BLOCKA\%Q22}
    string sID = "NetOut22"
    string sName = "NetOut22"
  [NetOut23]
    bool bActive
    bool bEnable = true
    dio dDio = {link=ApplicomIO-1\TOPIC1_A-BLOCKA\%Q23}
    string sID = "NetOut23"
    string sName = "NetOut23"
  [NetOut24]
    bool bActive
    bool bEnable = true
    dio dDio = {link=ApplicomIO-1\TOPIC1_A-BLOCKA\%Q24}
    string sID = "NetOut24"
    string sName = "NetOut24"
  [NetOut25]
    bool bActive
    bool bEnable = true
    dio dDio = {link=ApplicomIO-1\TOPIC1_A-BLOCKA\%Q25}
    string sID = "NetOut25"
    string sName = "NetOut25"
  [NetOut26]
    bool bActive
    bool bEnable = true
    dio dDio = {link=ApplicomIO-1\TOPIC1_A-BLOCKA\%Q26}
    string sID = "NetOut26"
    string sName = "NetOut26"
  [NetOut27]
    bool bActive
    bool bEnable = true
    dio dDio = {link=ApplicomIO-1\TOPIC1_A-BLOCKA\%Q27}
    string sID = "NetOut27"
    string sName = "NetOut27"
  [NetOut28]
    bool bActive
    bool bEnable = true
    dio dDio = {link=ApplicomIO-1\TOPIC1_A-BLOCKA\%Q28}
    string sID = "NetOut28"
    string sName = "NetOut28"
  [NetOut29]
    bool bActive
    bool bEnable = true
    dio dDio = {link=ApplicomIO-1\TOPIC1_A-BLOCKA\%Q29}
    string sID = "NetOut29"
    string sName = "NetOut29"
  [NetOut30]
    bool bActive
    bool bEnable = true
    dio dDio = {link=ApplicomIO-1\TOPIC1_A-BLOCKA\%Q30}
    string sID = "NetOut30"
    string sName = "NetOut30"
  [NetOut31]
    bool bActive
    bool bEnable = true
    dio dDio = {link=ApplicomIO-1\TOPIC1_A-BLOCKA\%Q31}
    string sID = "NetOut31"
    string sName = "NetOut31"
  [NetOut32]
    bool bActive
    bool bEnable = true
    dio dDio = {link=ApplicomIO-1\TOPIC1_A-BLOCKA\%Q32}
    string sID = "NetOut32"
    string sName = "NetOut32"
  [NetOut33]
    bool bActive
    bool bEnable = true
    dio dDio = {link=ApplicomIO-1\TOPIC1_A-BLOCKA\%Q33}
    string sID = "NetOut33"
    string sName = "NetOut33"
  [NetOut34]
    bool bActive
    bool bEnable = true
    dio dDio = {link=ApplicomIO-1\TOPIC1_A-BLOCKA\%Q34}
    string sID = "NetOut34"
    string sName = "NetOut34"
  [NetOut35]
    bool bActive
    bool bEnable = true
    dio dDio = {link=ApplicomIO-1\TOPIC1_A-BLOCKA\%Q35}
    string sID = "NetOut35"
    string sName = "NetOut35"
  [NetOut36]
    bool bActive
    bool bEnable = true
    dio dDio = {link=ApplicomIO-1\TOPIC1_A-BLOCKA\%Q36}
    string sID = "NetOut36"
    string sName = "NetOut36"
  [NetOut37]
    bool bActive
    bool bEnable = true
    dio dDio = {link=ApplicomIO-1\TOPIC1_A-BLOCKA\%Q37}
    string sID = "NetOut37"
    string sName = "NetOut37"
  [NetOut38]
    bool bActive
    bool bEnable = true
    dio dDio = {link=ApplicomIO-1\TOPIC1_A-BLOCKA\%Q38}
    string sID = "NetOut38"
    string sName = "NetOut38"
  [NetOut39]
    bool bActive
    bool bEnable = true
    dio dDio = {link=ApplicomIO-1\TOPIC1_A-BLOCKA\%Q39}
    string sID = "NetOut39"
    string sName = "NetOut39"
  [NetOut40]
    bool bActive
    bool bEnable = true
    dio dDio = {link=ApplicomIO-1\TOPIC1_A-BLOCKA\%Q40}
    string sID = "NetOut40"
    string sName = "NetOut40"
  [NetOut41]
    bool bActive
    bool bEnable = true
    dio dDio = {link=ApplicomIO-1\TOPIC1_A-BLOCKA\%Q41}
    string sID = "NetOut41"
    string sName = "NetOut41"
  [NetOut42]
    bool bActive
    bool bEnable = true
    dio dDio = {link=ApplicomIO-1\TOPIC1_A-BLOCKA\%Q42}
    string sID = "NetOut42"
    string sName = "NetOut42"
  [NetOut43]
    bool bActive
    bool bEnable = true
    dio dDio = {link=ApplicomIO-1\TOPIC1_A-BLOCKA\%Q43}
    string sID = "NetOut43"
    string sName = "NetOut43"
  [NetOut44]
    bool bActive
    bool bEnable = true
    dio dDio = {link=ApplicomIO-1\TOPIC1_A-BLOCKA\%Q44}
    string sID = "NetOut44"
    string sName = "NetOut44"
  [NetOut45]
    bool bActive
    bool bEnable = true
    dio dDio = {link=ApplicomIO-1\TOPIC1_A-BLOCKA\%Q45}
    string sID = "NetOut45"
    string sName = "NetOut45"
  [NetOut46]
    bool bActive
    bool bEnable = true
    dio dDio = {link=ApplicomIO-1\TOPIC1_A-BLOCKA\%Q46}
    string sID = "NetOut46"
